TYPE ST_DigitalInputParCmd :
STRUCT
    Reserved : BOOL; // passive monitor: physical four-structure contract, no command payload
END_STRUCT
END_TYPE

(* stored: Version 1.1.0.1, ProductVersion 3.1.4024.12
   DUT ST_DigitalInputParCmd: Id {846e57f1-9271-4c9c-8600-217a72426b15} *)
